INTERFACE ITF_EspHost

METHOD CyclicUpdate : BOOL
VAR_INPUT
END_VAR
END_METHOD

METHOD GetDataBuffer : BOOL
VAR_INPUT
	Address	: REFERENCE TO PVOID;
	Size	: REFERENCE TO UDINT;
END_VAR
END_METHOD

METHOD GetLastReceivedIp : T_IPv4Addr
VAR_INPUT
END_VAR
END_METHOD

METHOD GetFirstReceivedTimestamp : ULINT
VAR_INPUT
END_VAR
END_METHOD

METHOD GetLastReceivedTimestamp : ULINT
VAR_INPUT
END_VAR
END_METHOD

METHOD GetMetadata : EspPacketHeader
VAR_INPUT
END_VAR
END_METHOD

METHOD GetPacketToSend : BOOL
VAR_INPUT
	Address	: REFERENCE TO PVOID;
	Size	: REFERENCE TO UDINT;
END_VAR
END_METHOD

METHOD GetPacketsReceived : ULINT
VAR_INPUT
END_VAR
END_METHOD

METHOD GetSystemInfo : EspSystemInfo
VAR_INPUT
END_VAR
END_METHOD

METHOD IsOnline : BOOL
VAR_INPUT
	Timeout100Ns	: ULINT;
END_VAR
END_METHOD

METHOD SetLastReceivedIp : BOOL
VAR_INPUT
	IpAddress	: T_IPv4Addr;
END_VAR
END_METHOD

METHOD SetPacketType : BOOL
VAR_INPUT
	PacketType	: BYTE;
END_VAR
END_METHOD

METHOD SetUID : BOOL
VAR_INPUT
	UID	: ULINT;
END_VAR
END_METHOD

METHOD UpdateMetadata : BOOL
VAR_INPUT
	Data	: EspPacketHeader;
END_VAR
END_METHOD

METHOD UpdateSystemInfo : BOOL
VAR_INPUT
	PayloadAddress	: PVOID;
	PayloadLength	: UINT;
END_VAR
END_METHOD

END_INTERFACE

(* stored: Version 1.1.0.1
   Itf ITF_EspHost: Id {abc0fd08-8675-407a-972a-8d22e58329f4}
   Method CyclicUpdate: Id {d54f9482-e9a0-4911-8758-6dc451e9417d}
   Method GetDataBuffer: Id {8da7ba6e-02ea-4334-8c55-9511c73189e8}
   Method GetLastReceivedIp: Id {b7e8a521-5b32-47c4-9229-b8ba2629d06e}
   Method GetFirstReceivedTimestamp: Id {e2189e05-1af7-4574-83c8-0c4f2e0b8d78}
   Method GetLastReceivedTimestamp: Id {0e25293d-26cc-4bf6-a81d-2a85d9d14a0d}
   Method GetMetadata: Id {092453f9-bdfc-451c-9a98-2b2b149e9714}
   Method GetPacketToSend: Id {abdcee37-5220-45a6-94c7-6a0aa945a685}
   Method GetPacketsReceived: Id {b7b940a6-3a3a-4eb4-99a5-9776e074dc9b}
   Method GetSystemInfo: Id {0e558af3-cb9d-4c9e-a942-3e9bd778219a}
   Method IsOnline: Id {c3927e27-7d07-40de-bb17-0055d95c1d8c}
   Method SetLastReceivedIp: Id {5a73b017-dcc1-4b95-b1f5-a4c33fa6b29b}
   Method SetPacketType: Id {e3c007f5-3d89-4e0e-a60d-918d2cfb4649}
   Method SetUID: Id {be2bad33-45cb-4a7d-89f3-5afa2d7f7753}
   Method UpdateMetadata: Id {f63b2cb9-24e9-4405-8a20-3118827fa9aa}
   Method UpdateSystemInfo: Id {ef7b2959-420b-4ef2-b5ea-8c3599fef9a5} *)
